// TIA Portal project "红黄绿等" (V16)

(* hardware
DEVICE "HMI_1"  KTP700 Basic PN
   slot 0: "HMI_1"  KTP700 Basic PN  6AV2 123-2GB03-0AX0  16.0.0.0
   slot 1: "HMI_RT_1"  KTP700 Basic PN  6AV2 123-2GB03-0AX0  16.0.0.0
   slot 5: "HMI_1.IE_CP_1"  PROFINET Interface  16.0.0.0
      slot 1: "PROFINET Interface_1"  PROFINET Interface
         slot 1: "Port_1"  Port
DEVICE "S7-1200 station_1"  S7-1200 Station
   slot 0: "Rack_0"  S7-1200 Rack  Rack  V1.0
   slot 1: "PLC_1"  CPU 1212C DC/DC/DC  6ES7 212-1AE40-0XB0  V4.2
   slot 2: "DI 16/DQ 16x24VDC_1"  6ES7 223-1BL32-0XB0  V2.0
DEVICE "S7-1200 station_2"  S7-1200 Station
   slot 0: "Rack_0"  S7-1200 Rack  Rack  V1.0
   slot 1: "PLC_2"  CPU 1212C DC/DC/DC  6ES7 212-1AE40-0XB0  V4.2
   slot 2: "DI 16/DQ 16x24VDC_1"  6ES7 223-1BL32-0XB0  V2.0
*)

// ===== PLC "PLC_1"  CPU 1212C DC/DC/DC =====

VAR_GLOBAL   // PLC tag table "默认变量表"
   "System_Byte" AT %MB1 : Byte;
   "FirstScan" AT %M1.0 : Bool;
   "DiagStatusUpdate" AT %M1.1 : Bool;
   "AlwaysTRUE" AT %M1.2 : Bool;
   "AlwaysFALSE" AT %M1.3 : Bool;
   "Tag_1" AT %M8.1 : Bool;
   "Tag_3" AT %MD90 : Real;
   "Tag_4" AT %MD80 : Real;
END_VAR

VAR_GLOBAL   // PLC tag table "io表"
   "x轴脉冲" AT %Q0.0 : Bool;
   "x轴方向" AT %Q0.1 : Bool;
   "z轴脉冲" AT %Q0.2 : Bool;
   "z轴方向" AT %Q0.3 : Bool;
   "x轴前限位" AT %I0.0 : Bool;
   "x轴原点" AT %I0.1 : Bool;
   "x轴后限位" AT %I0.2 : Bool;
   "z轴上限位" AT %I0.3 : Bool;
   "z轴原点" AT %I0.4 : Bool;
   "z轴下限位" AT %I0.5 : Bool;
   "输送线A右传感器" AT %I1.0 : Bool;
   "输送线A左传感器" AT %I1.1 : Bool;
   "启动" AT %I1.4 : Bool;
   "复位" AT %I1.5 : Bool;
   "急停" AT %I1.6 : Bool;
   "单机/联动" AT %I1.7 : Bool;
   "旋转气缸左转" AT %I2.0 : Bool;
   "旋转气缸右转" AT %I2.1 : Bool;
   "伸出前限位" AT %I2.2 : Bool;
   "伸出后限位" AT %I2.3 : Bool;
   "黄灯" AT %Q1.0 : Bool;
   "红灯" AT %Q1.2 : Bool;
   "气缸左旋" AT %Q1.4 : Bool;
   "气缸右旋" AT %Q1.5 : Bool;
   "气缸伸缩" AT %Q1.6 : Bool;
   "气缸夹紧" AT %Q1.7 : Bool;
   "输送带A正转" AT %Q2.0 : Bool;
   "输送带A反转" AT %Q2.1 : Bool;
   "手自动切换" AT %M2.6 : Bool;
   "自动启动按钮" AT %M2.7 : Bool;
   "x轴前进-触点" AT %M6.0 : Bool;
   "x轴后退-触点" AT %M6.1 : Bool;
   "z轴下移-触点" AT %M6.2 : Bool;
   "z轴上移-触点" AT %M6.3 : Bool;
   "x轴前进" AT %M7.0 : Bool;
   "x轴后退" AT %M7.1 : Bool;
   "x轴回原点" AT %M7.2 : Bool;
   "z轴上移" AT %M7.3 : Bool;
   "z轴下移" AT %M7.4 : Bool;
   "z轴回原点" AT %M7.5 : Bool;
   "x轴启动标志位" AT %M2.0 : Bool;
   "x轴完成标志位" AT %M2.1 : Bool;
   "z轴启动标志位" AT %M2.2 : Bool;
   "z轴完成标志位" AT %M2.3 : Bool;
   "x轴回原点(1)" AT %M2.4 : Bool;
   "z轴回原点(1)" AT %M2.5 : Bool;
   "启动整个程序" AT %M5.0 : Bool;
   "tag_2" AT %M5.2 : Bool;
   "自动模式" AT %M5.3 : Bool;
   "x轴取料移动标志" AT %M3.0 : Bool;
   "tag_5" AT %M20.0 : Bool;
   "z轴取料移动标志位" AT %M3.1 : Bool;
   "tag_7" AT %M20.1 : Bool;
   "x轴定位数据" AT %MD30 : Real;
   "z轴定位数据" AT %MD40 : Real;
   "启动气缸左旋标志位" AT %M3.2 : Bool;
   "启动气缸伸缩标志位" AT %M3.3 : Bool;
   "启动气缸夹取标志位" AT %M3.4 : Bool;
   "z轴上升标志位" AT %M3.5 : Bool;
   "tag_12" AT %M20.2 : Bool;
   "气缸回缩标志位" AT %M3.6 : Bool;
   "气缸右旋标志位" AT %M3.7 : Bool;
   "x轴启动放料位" AT %M4.0 : Bool;
   "tag_16" AT %M20.3 : Bool;
   "z轴上升到放料位" AT %M4.1 : Bool;
   "tag_18" AT %M20.4 : Bool;
   "气缸伸出放料标志位" AT %M4.2 : Bool;
   "气缸放松放料标志位" AT %M4.3 : Bool;
   "tag_21" AT %M4.4 : Bool;
   "X轴报错复位" AT %M7.6 : Bool;
   "z轴报错复位" AT %M7.7 : Bool;
   "tag_22" AT %MD50 : Real;
   "tag_23" AT %MD60 : Real;
   "tag_24" AT %MD70 : Real;
   "绿灯" AT %Q1.1 : Bool;
END_VAR

// folder: System blocks/Program resources

DATA_BLOCK "T1"   // DB3
{ S7_Optimized_Access := 'TRUE' }
AUTHOR : Simatic
FAMILY : IEC
NAME : IEC_TMR
VERSION : 1.0
// stored: InstanceOfName IEC_TIMER
"IEC_TIMER"
BEGIN
END_DATA_BLOCK

DATA_BLOCK "T2"   // DB4
{ S7_Optimized_Access := 'TRUE' }
AUTHOR : Simatic
FAMILY : IEC
NAME : IEC_TMR
VERSION : 1.0
// stored: InstanceOfName IEC_TIMER
"IEC_TIMER"
BEGIN
END_DATA_BLOCK

DATA_BLOCK "T3"   // DB5
{ S7_Optimized_Access := 'TRUE' }
AUTHOR : Simatic
FAMILY : IEC
NAME : IEC_TMR
VERSION : 1.0
// stored: InstanceOfName IEC_TIMER
"IEC_TIMER"
BEGIN
END_DATA_BLOCK

DATA_BLOCK "T4"   // DB6
{ S7_Optimized_Access := 'TRUE' }
AUTHOR : Simatic
FAMILY : IEC
NAME : IEC_TMR
VERSION : 1.0
// stored: InstanceOfName IEC_TIMER
"IEC_TIMER"
BEGIN
END_DATA_BLOCK

DATA_BLOCK "T5"   // DB7
{ S7_Optimized_Access := 'TRUE' }
AUTHOR : Simatic
FAMILY : IEC
NAME : IEC_TMR
VERSION : 1.0
// stored: InstanceOfName IEC_TIMER
"IEC_TIMER"
BEGIN
END_DATA_BLOCK

DATA_BLOCK "T7"   // DB8
{ S7_Optimized_Access := 'TRUE' }
AUTHOR : Simatic
FAMILY : IEC
NAME : IEC_TMR
VERSION : 1.0
// stored: InstanceOfName IEC_TIMER
"IEC_TIMER"
BEGIN
END_DATA_BLOCK

DATA_BLOCK "T6"   // DB9
{ S7_Optimized_Access := 'TRUE' }
AUTHOR : Simatic
FAMILY : IEC
NAME : IEC_TMR
VERSION : 1.0
// stored: InstanceOfName IEC_TIMER
"IEC_TIMER"
BEGIN
END_DATA_BLOCK

DATA_BLOCK "T8"   // DB10
{ S7_Optimized_Access := 'TRUE' }
AUTHOR : Simatic
FAMILY : IEC
NAME : IEC_TMR
VERSION : 1.0
// stored: InstanceOfName IEC_TIMER
"IEC_TIMER"
BEGIN
END_DATA_BLOCK

DATA_BLOCK "T9"   // DB11
{ S7_Optimized_Access := 'TRUE' }
AUTHOR : Simatic
FAMILY : IEC
NAME : IEC_TMR
VERSION : 1.0
// stored: InstanceOfName IEC_TIMER
"IEC_TIMER"
BEGIN
END_DATA_BLOCK

DATA_BLOCK "T10"   // DB12
{ S7_Optimized_Access := 'TRUE' }
AUTHOR : Simatic
FAMILY : IEC
NAME : IEC_TMR
VERSION : 1.0
// stored: InstanceOfName IEC_TIMER
"IEC_TIMER"
BEGIN
END_DATA_BLOCK

DATA_BLOCK "T11"   // DB13
{ S7_Optimized_Access := 'TRUE' }
AUTHOR : Simatic
FAMILY : IEC
NAME : IEC_TMR
VERSION : 1.0
// stored: InstanceOfName IEC_TIMER
"IEC_TIMER"
BEGIN
END_DATA_BLOCK

DATA_BLOCK "T12"   // DB14
{ S7_Optimized_Access := 'TRUE' }
AUTHOR : Simatic
FAMILY : IEC
NAME : IEC_TMR
VERSION : 1.0
// stored: InstanceOfName IEC_TIMER
"IEC_TIMER"
BEGIN
END_DATA_BLOCK

DATA_BLOCK "T13"   // DB15
{ S7_Optimized_Access := 'TRUE' }
AUTHOR : Simatic
FAMILY : IEC
NAME : IEC_TMR
VERSION : 1.0
// stored: InstanceOfName IEC_TIMER
"IEC_TIMER"
BEGIN
END_DATA_BLOCK

DATA_BLOCK "IEC_Timer_0_DB"   // DB28
{ S7_Optimized_Access := 'TRUE' }
AUTHOR : Simatic
FAMILY : IEC
NAME : IEC_TMR
VERSION : 1.0
// stored: InstanceOfName IEC_TIMER
"IEC_TIMER"
BEGIN
END_DATA_BLOCK

// folder: (top level)

DATA_BLOCK "轴_1"   // DB1, Motion_DB
{ S7_Optimized_Access := 'TRUE' }
AUTHOR : SIMATIC
FAMILY : BasicMC
NAME : TO_PosAx
VERSION : 6.0
// stored: InstanceOfName TO_PositioningAxis
"TO_PositioningAxis"
BEGIN
   // Axis.HomingReferencePointSwitch_AddressCU = %I0.1
   // Axis.LengthUnitNormalized.Distance = 1013
   // Axis.PositionLimitsMax_AddressCU = %I0.2
   // Axis.PositionLimitsMin_AddressCU = %I0.0
   // Axis.DirectionOutputEnabledCU = TRUE
   // Axis.OnlinePtoModeCU = 16#0000_0002
   // Axis.SelectedChannel2EnumCU = %Q0.1
   // Axis.SelectedChannel1EnumCU = %Q0.0
   // Pulse.MinDeltaDeltaFrequencyCU = 0.004
   // Pulse.MaxDeltaDeltaFrequencyCU = 1.0E+10
   // Pulse.MinDeltaFrequencyCU = 0.005
   // Pulse.MaxDeltaFrequencyCU = 9.5E+9
   // Pulse.MinFrequencyCU = 1.0
   // Pulse.MaxFrequencyCU = 100000.0
   // Pulse.OutputSourceCU = 16#0000_0000
   // Axis.SelectPTO = 0
END_DATA_BLOCK

DATA_BLOCK "轴_2"   // DB2, Motion_DB
{ S7_Optimized_Access := 'TRUE' }
AUTHOR : SIMATIC
FAMILY : BasicMC
NAME : TO_PosAx
VERSION : 6.0
// stored: InstanceOfName TO_PositioningAxis
"TO_PositioningAxis"
BEGIN
   // Axis.HomingReferencePointSwitch_AddressCU = %I0.4
   // Axis.LengthUnitNormalized.Distance = 1013
   // Axis.PositionLimitsMax_AddressCU = %I0.5
   // Axis.PositionLimitsMin_AddressCU = %I0.3
   // Axis.DirectionOutputEnabledCU = TRUE
   // Axis.OnlinePtoModeCU = 16#0000_0002
   // Axis.SelectedChannel2EnumCU = %Q0.3
   // Axis.SelectedChannel1EnumCU = %Q0.2
   // Pulse.MinDeltaDeltaFrequencyCU = 0.004
   // Pulse.MaxDeltaDeltaFrequencyCU = 1.0E+10
   // Pulse.MinDeltaFrequencyCU = 0.005
   // Pulse.MaxDeltaFrequencyCU = 9.5E+9
   // Pulse.MinFrequencyCU = 1.0
   // Pulse.MaxFrequencyCU = 100000.0
   // Pulse.OutputSourceCU = 16#0000_0000
   // Axis.SelectPTO = 1
   // Axis.OnlinePtoIndexCU = 1
END_DATA_BLOCK

FUNCTION "电机运转" : Void   // FC1, LAD
{ S7_Optimized_Access := 'TRUE' }
VERSION : 0.1
BEGIN

REGION Network 1: 启动两个电机轴
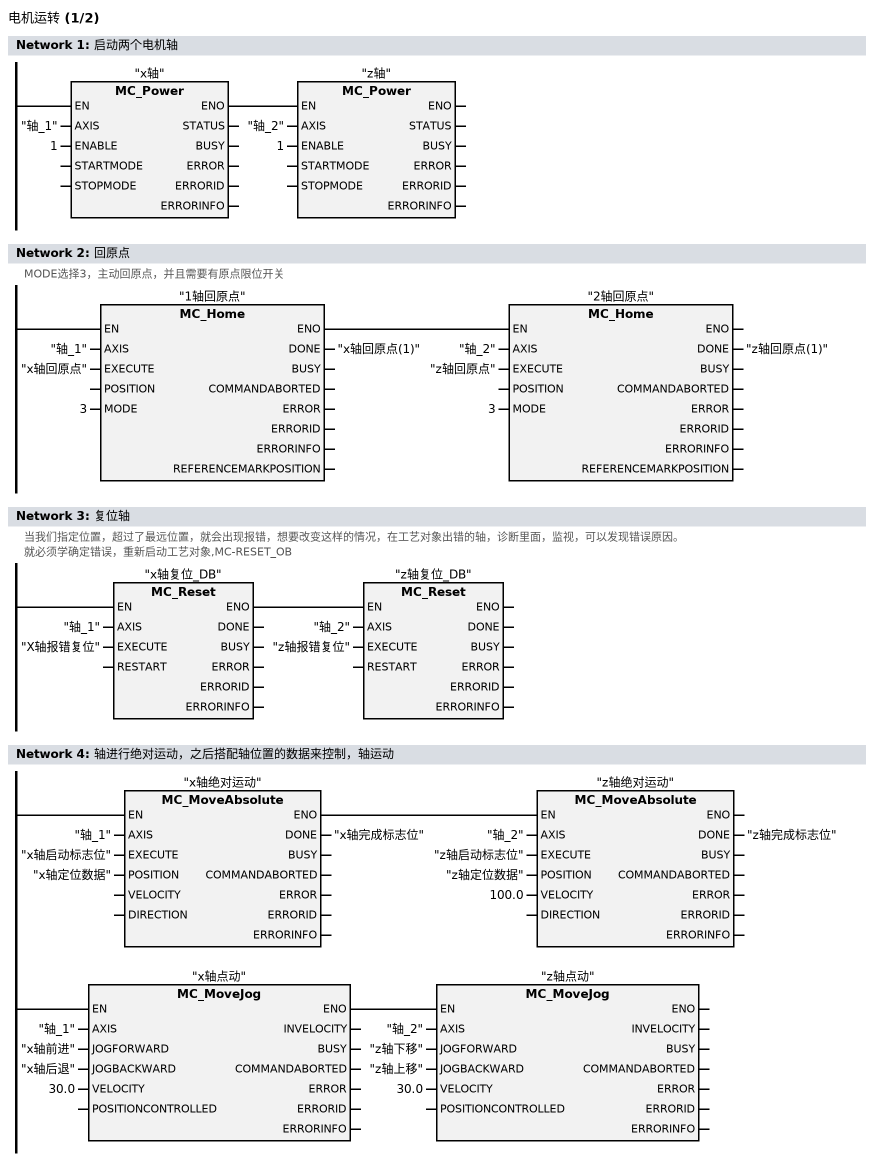
   // ENO of a box is taken as its EN; it also drops when the box reports an error
   "x轴"(Axis := "轴_1", Enable := 1);   // MC_Power
   "z轴"(Axis := "轴_2", Enable := 1);   // MC_Power
END_REGION

REGION Network 2: 回原点
   // MODE选择3，主动回原点，并且需要有原点限位开关
   // ENO of a box is taken as its EN; it also drops when the box reports an error
   "1轴回原点"(Axis := "轴_1", Execute := "x轴回原点", Mode := 3, Done => "x轴回原点(1)");   // MC_Home
   "2轴回原点"(Axis := "轴_2", Execute := "z轴回原点", Mode := 3, Done => "z轴回原点(1)");   // MC_Home
END_REGION

REGION Network 3: 复位轴
   // 当我们指定位置，超过了最远位置，就会出现报错，想要改变这样的情况，在工艺对象出错的轴，诊断里面，监视，可以发现错误原因。
   // 就必须学确定错误，重新启动工艺对象,MC-RESET_OB
   // ENO of a box is taken as its EN; it also drops when the box reports an error
   "x轴复位_DB"(Axis := "轴_1", Execute := "X轴报错复位");   // MC_Reset
   "z轴复位_DB"(Axis := "轴_2", Execute := "z轴报错复位");   // MC_Reset
END_REGION

REGION Network 4: 轴进行绝对运动，之后搭配轴位置的数据来控制，轴运动
   // ENO of a box is taken as its EN; it also drops when the box reports an error
   "x轴绝对运动"(Axis := "轴_1", Execute := "x轴启动标志位", Position := "x轴定位数据", Done => "x轴完成标志位");   // MC_MoveAbsolute
   "z轴绝对运动"(Axis := "轴_2", Execute := "z轴启动标志位", Position := "z轴定位数据", Velocity := 100.0, Done => "z轴完成标志位");   // MC_MoveAbsolute
   "x轴点动"(Axis := "轴_1", JogForward := "x轴前进", JogBackward := "x轴后退", Velocity := 30.0);   // MC_MoveJog
   "z轴点动"(Axis := "轴_2", JogForward := "z轴下移", JogBackward := "z轴上移", Velocity := 30.0);   // MC_MoveJog
END_REGION

REGION Network 5
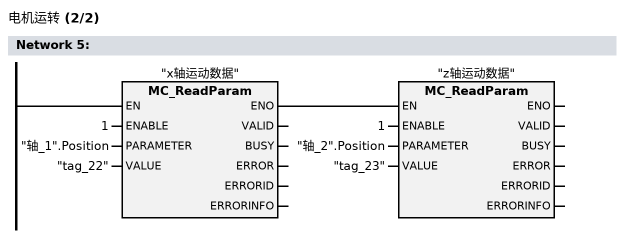
   // ENO of a box is taken as its EN; it also drops when the box reports an error
   "x轴运动数据"(Enable := 1, Parameter := "轴_1".Position, Value := "tag_22");   // MC_ReadParam
   "z轴运动数据"(Enable := 1, Parameter := "轴_2".Position, Value := "tag_23");   // MC_ReadParam
END_REGION
END_FUNCTION

ORGANIZATION_BLOCK "Main"   // OB1, LAD, ProgramCycle
TITLE = "Main Program Sweep (Cycle)"
{ S7_Optimized_Access := 'TRUE' }
VERSION : 0.1
   VAR_INPUT
      Initial_Call : Bool;   // Initial call of this OB
      Remanence : Bool;   // =True, if remanent data are available
   END_VAR
   VAR_TEMP   // added for the SCL form of the ladder/FBD networks
      _w1 : Bool;
      _w2 : Bool;
      _w3 : Bool;
   END_VAR
BEGIN

REGION Network 1: 初始化程序，并且启动程序
   // 利用M1.0达到首次循环，启动复位
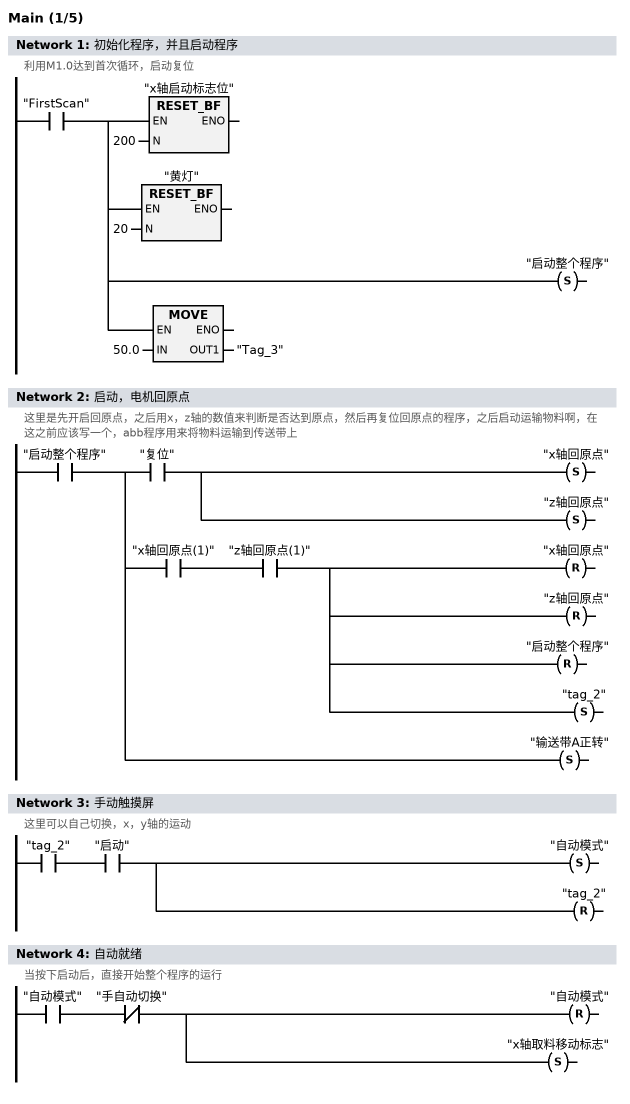
   // no SCL statement known for RBitfield: written as a call
   #_w1 := "FirstScan";
   IF #_w1 THEN
       RESET_BF(operand := "x轴启动标志位", n := 200);
       RESET_BF(operand := "黄灯", n := 20);
       "启动整个程序" := TRUE;
       "Tag_3" := 50.0;
   END_IF;
END_REGION

REGION Network 2: 启动，电机回原点
   // 这里是先开启回原点，之后用x，z轴的数值来判断是否达到原点，然后再复位回原点的程序，之后启动运输物料啊，在这之前应该写一个，abb程序用来将物料运输到传送带上
   RUNG wire#powerrail
      Contact( "启动整个程序" )
      wire#w1
      Contact( "复位" )
      wire#w2
      S_Coil( "x轴回原点" )
   END_RUNG
   RUNG wire#w2
      S_Coil( "z轴回原点" )
   END_RUNG
   RUNG wire#w1
      Contact( "x轴回原点(1)" )
      Contact( "z轴回原点(1)" )
      wire#w3
      R_Coil( "x轴回原点" )
   END_RUNG
   RUNG wire#w3
      R_Coil( "z轴回原点" )
   END_RUNG
   RUNG wire#w3
      R_Coil( "启动整个程序" )
   END_RUNG
   RUNG wire#w3
      S_Coil( "tag_2" )
   END_RUNG
   RUNG wire#w1
      S_Coil( "输送带A正转" )
   END_RUNG
   // the same network as SCL:
   IF "启动整个程序" AND "复位" THEN
       "x轴回原点" := TRUE;
       "z轴回原点" := TRUE;
   END_IF;
   IF "启动整个程序" AND "x轴回原点(1)" AND "z轴回原点(1)" THEN
       "x轴回原点" := FALSE;
       "z轴回原点" := FALSE;
   END_IF;
   #_w1 := "启动整个程序";
   #_w2 := "启动整个程序" AND "x轴回原点(1)" AND "z轴回原点(1)";
   IF #_w2 THEN
       "启动整个程序" := FALSE;
       "tag_2" := TRUE;
   END_IF;
   IF #_w1 THEN "输送带A正转" := TRUE; END_IF;
END_REGION

REGION Network 3: 手动触摸屏
   // 这里可以自己切换，x，y轴的运动
   RUNG wire#powerrail
      Contact( "tag_2" )
      Contact( "启动" )
      wire#w1
      S_Coil( "自动模式" )
   END_RUNG
   RUNG wire#w1
      R_Coil( "tag_2" )
   END_RUNG
   // the same network as SCL:
   IF "tag_2" AND "启动" THEN
       "自动模式" := TRUE;
       "tag_2" := FALSE;
   END_IF;
END_REGION

REGION Network 4: 自动就绪
   // 当按下启动后，直接开始整个程序的运行
   RUNG wire#powerrail
      Contact( "自动模式" )
      I_Contact( "手自动切换" )
      wire#w1
      R_Coil( "自动模式" )
   END_RUNG
   RUNG wire#w1
      S_Coil( "x轴取料移动标志" )
   END_RUNG
   // the same network as SCL:
   #_w1 := "自动模式" AND NOT "手自动切换";
   IF #_w1 THEN
       "自动模式" := FALSE;
       "x轴取料移动标志" := TRUE;
   END_IF;
END_REGION

REGION Network 5: x轴取料
   // 此处对应传送带上的传感器，限位开关感应到物料,，输送带停止输送
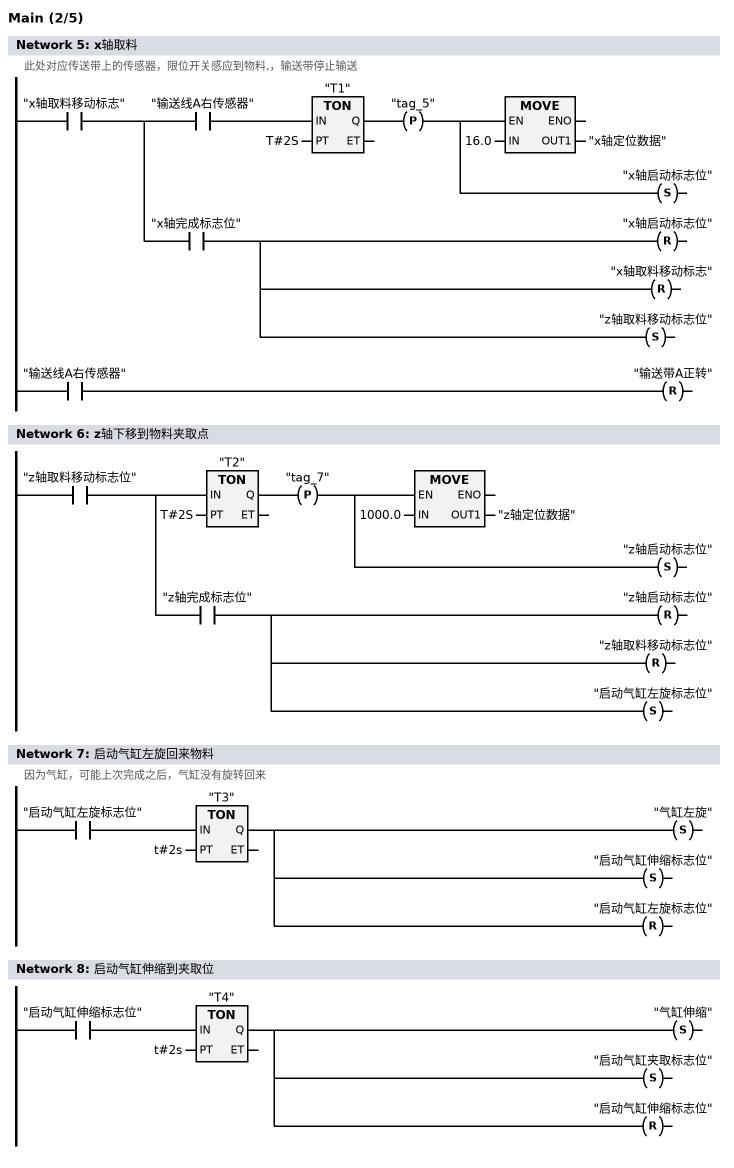
   "T1".TON(IN := "x轴取料移动标志" AND "输送线A右传感器", PT := T#2S);
   #_w1 := "T1".Q AND NOT "tag_5";   // rising edge
   "tag_5" := "T1".Q;
   IF #_w1 THEN
       "x轴定位数据" := 16.0;
       "x轴启动标志位" := TRUE;
   END_IF;
   IF "x轴取料移动标志" AND "x轴完成标志位" THEN "x轴启动标志位" := FALSE; END_IF;
   #_w2 := "x轴取料移动标志" AND "x轴完成标志位";
   IF #_w2 THEN
       "x轴取料移动标志" := FALSE;
       "z轴取料移动标志位" := TRUE;
   END_IF;
   IF "输送线A右传感器" THEN "输送带A正转" := FALSE; END_IF;
END_REGION

REGION Network 6: z轴下移到物料夹取点
   "T2".TON(IN := "z轴取料移动标志位", PT := T#2S);
   #_w1 := "T2".Q AND NOT "tag_7";   // rising edge
   "tag_7" := "T2".Q;
   IF #_w1 THEN
       "z轴定位数据" := 1000.0;
       "z轴启动标志位" := TRUE;
   END_IF;
   IF "z轴取料移动标志位" AND "z轴完成标志位" THEN "z轴启动标志位" := FALSE; END_IF;
   #_w2 := "z轴取料移动标志位" AND "z轴完成标志位";
   IF #_w2 THEN
       "z轴取料移动标志位" := FALSE;
       "启动气缸左旋标志位" := TRUE;
   END_IF;
END_REGION

REGION Network 7: 启动气缸左旋回来物料
   // 因为气缸，可能上次完成之后，气缸没有旋转回来
   "T3".TON(IN := "启动气缸左旋标志位", PT := t#2s);
   IF "T3".Q THEN
       "气缸左旋" := TRUE;
       "启动气缸伸缩标志位" := TRUE;
       "启动气缸左旋标志位" := FALSE;
   END_IF;
END_REGION

REGION Network 8: 启动气缸伸缩到夹取位
   "T4".TON(IN := "启动气缸伸缩标志位", PT := t#2s);
   IF "T4".Q THEN
       "气缸伸缩" := TRUE;
       "启动气缸夹取标志位" := TRUE;
       "启动气缸伸缩标志位" := FALSE;
   END_IF;
END_REGION

REGION Network 9: 启动气缸夹取
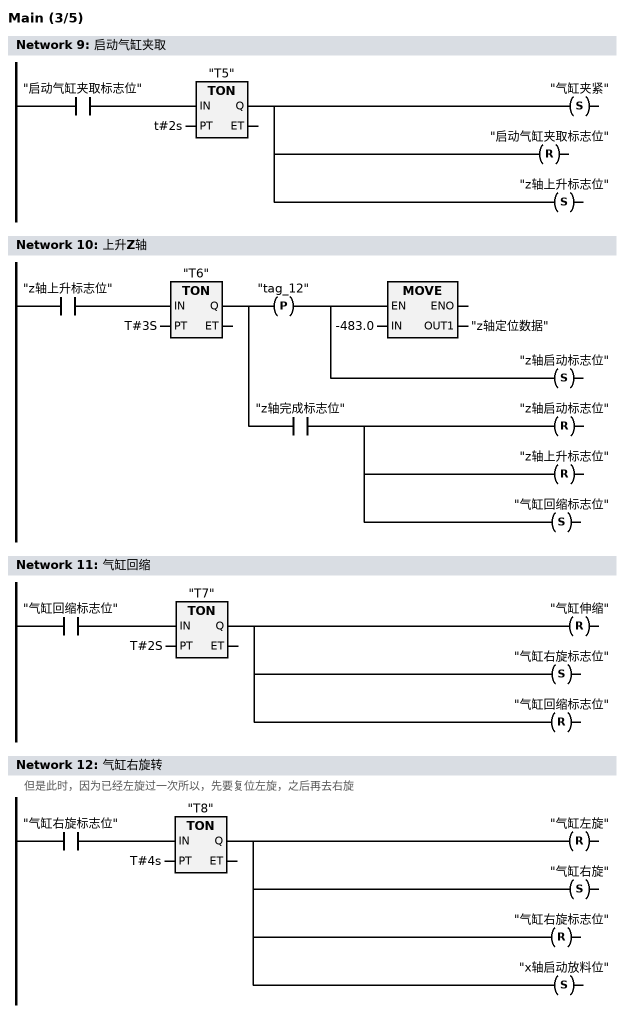
   "T5".TON(IN := "启动气缸夹取标志位", PT := t#2s);
   IF "T5".Q THEN
       "气缸夹紧" := TRUE;
       "启动气缸夹取标志位" := FALSE;
       "z轴上升标志位" := TRUE;
   END_IF;
END_REGION

REGION Network 10: 上升Z轴
   "T6".TON(IN := "z轴上升标志位", PT := T#3S);
   #_w1 := "T6".Q AND NOT "tag_12";   // rising edge
   "tag_12" := "T6".Q;
   IF #_w1 THEN
       "z轴定位数据" := -483.0;
       "z轴启动标志位" := TRUE;
   END_IF;
   IF "T6".Q AND "z轴完成标志位" THEN
       "z轴启动标志位" := FALSE;
       "z轴上升标志位" := FALSE;
       "气缸回缩标志位" := TRUE;
   END_IF;
END_REGION

REGION Network 11: 气缸回缩
   "T7".TON(IN := "气缸回缩标志位", PT := T#2S);
   IF "T7".Q THEN
       "气缸伸缩" := FALSE;
       "气缸右旋标志位" := TRUE;
       "气缸回缩标志位" := FALSE;
   END_IF;
END_REGION

REGION Network 12: 气缸右旋转
   // 但是此时，因为已经左旋过一次所以，先要复位左旋，之后再去右旋
   "T8".TON(IN := "气缸右旋标志位", PT := T#4s);
   IF "T8".Q THEN
       "气缸左旋" := FALSE;
       "气缸右旋" := TRUE;
       "气缸右旋标志位" := FALSE;
       "x轴启动放料位" := TRUE;
   END_IF;
END_REGION

REGION Network 13: x轴移动到放料位
   // 我对于x轴来说，每排放3个，
   // 所以当我想要进行循环的时候，我可以写一个递增的数据，每当x移动3次之后
   // 就在z轴上升的程序里面，进行一次加法/减法计算
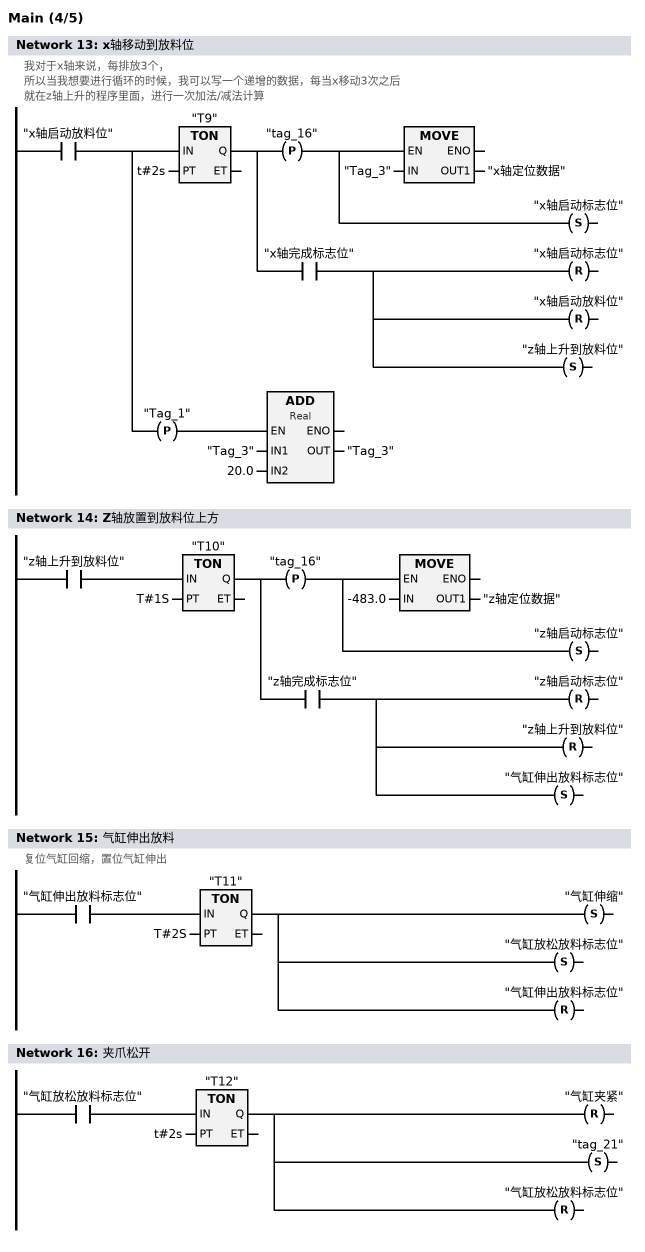
   "T9".TON(IN := "x轴启动放料位", PT := t#2s);
   #_w1 := "T9".Q AND NOT "tag_16";   // rising edge
   "tag_16" := "T9".Q;
   IF #_w1 THEN
       "x轴定位数据" := "Tag_3";
       "x轴启动标志位" := TRUE;
   END_IF;
   IF "T9".Q AND "x轴完成标志位" THEN "x轴启动标志位" := FALSE; END_IF;
   #_w2 := "x轴启动放料位";
   IF "T9".Q AND "x轴完成标志位" THEN
       "x轴启动放料位" := FALSE;
       "z轴上升到放料位" := TRUE;
   END_IF;
   #_w3 := #_w2 AND NOT "Tag_1";   // rising edge
   "Tag_1" := #_w2;
   IF #_w3 THEN "Tag_3" := "Tag_3" + 20.0; END_IF;
END_REGION

REGION Network 14: Z轴放置到放料位上方
   "T10".TON(IN := "z轴上升到放料位", PT := T#1S);
   #_w1 := "T10".Q AND NOT "tag_16";   // rising edge
   "tag_16" := "T10".Q;
   IF #_w1 THEN
       "z轴定位数据" := -483.0;
       "z轴启动标志位" := TRUE;
   END_IF;
   IF "T10".Q AND "z轴完成标志位" THEN
       "z轴启动标志位" := FALSE;
       "z轴上升到放料位" := FALSE;
       "气缸伸出放料标志位" := TRUE;
   END_IF;
END_REGION

REGION Network 15: 气缸伸出放料
   // 复位气缸回缩，置位气缸伸出
   "T11".TON(IN := "气缸伸出放料标志位", PT := T#2S);
   IF "T11".Q THEN
       "气缸伸缩" := TRUE;
       "气缸放松放料标志位" := TRUE;
       "气缸伸出放料标志位" := FALSE;
   END_IF;
END_REGION

REGION Network 16: 夹爪松开
   "T12".TON(IN := "气缸放松放料标志位", PT := t#2s);
   IF "T12".Q THEN
       "气缸夹紧" := FALSE;
       "tag_21" := TRUE;
       "气缸放松放料标志位" := FALSE;
   END_IF;
END_REGION

REGION Network 17: 结束复位
   // 如果要进行循环，此处应该重新置位
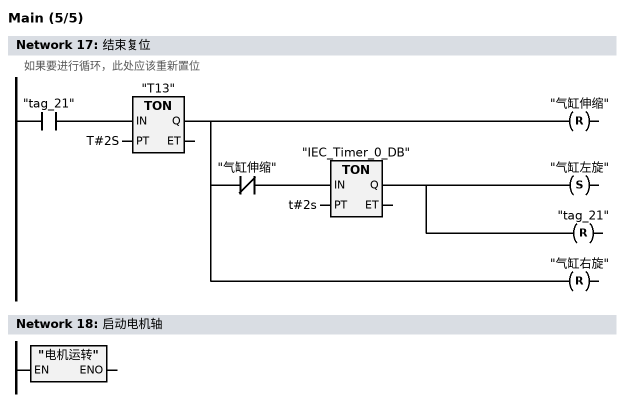
   "T13".TON(IN := "tag_21", PT := T#2S);
   IF "T13".Q THEN "气缸伸缩" := FALSE; END_IF;
   "IEC_Timer_0_DB".TON(IN := "T13".Q AND NOT "气缸伸缩", PT := t#2s);
   IF "IEC_Timer_0_DB".Q THEN
       "气缸左旋" := TRUE;
       "tag_21" := FALSE;
   END_IF;
   IF "T13".Q THEN "气缸右旋" := FALSE; END_IF;
END_REGION

REGION Network 18: 启动电机轴
   RUNG wire#powerrail
      "电机运转"()
   END_RUNG
   // the same network as SCL:
   "电机运转"();
END_REGION
END_ORGANIZATION_BLOCK

// ===== PLC "PLC_2"  CPU 1212C DC/DC/DC =====

VAR_GLOBAL   // PLC tag table "默认变量表"
   "Tag_1" AT %I1.4 : Bool;
   "Tag_2" AT %I1.5 : Bool;
   "Tag_3" AT %Q1.1 : Bool;
   "x轴脉冲" AT %Q0.0 : Bool;
   "x轴方向" AT %Q0.1 : Bool;
   "轴_1_LowHwLimitSwitch" AT %I0.0 : Bool;
   "轴_1_HighHwLimitSwitch" AT %I0.2 : Bool;
   "轴_1_归位开关" AT %I0.1 : Bool;
   "z轴脉冲" AT %Q0.2 : Bool;
   "z轴方向" AT %Q0.3 : Bool;
   "轴_2_LowHwLimitSwitch" AT %I0.3 : Bool;
   "轴_2_HighHwLimitSwitch" AT %I0.5 : Bool;
   "轴_2_归位开关" AT %I0.4 : Bool;
END_VAR

ORGANIZATION_BLOCK "Main"   // OB1, LAD, ProgramCycle
TITLE = "Main Program Sweep (Cycle)"
{ S7_Optimized_Access := 'TRUE' }
VERSION : 0.1
   VAR_INPUT
      Initial_Call : Bool;   // Initial call of this OB
      Remanence : Bool;   // =True, if remanent data are available
   END_VAR
BEGIN

REGION Network 1
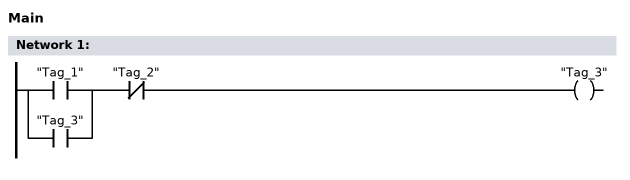
   RUNG wire#powerrail
      Contact( "Tag_1" )
      wire#w1
      I_Contact( "Tag_2" )
      Coil( "Tag_3" )
   END_RUNG
   RUNG wire#powerrail
      Contact( "Tag_3" )
   END_RUNG wire#w1
   // the same network as SCL:
   "Tag_3" := ("Tag_1" OR "Tag_3") AND NOT "Tag_2";
END_REGION
END_ORGANIZATION_BLOCK

(* ===== HMI "HMI_RT_1" =====
system functions are stored by id; their names below are inferred from use
connection "HMI_连接_1": ETHERNET, SMART_S7_1200_OMS

HMI tags "默认变量表"
   "Tag_ScreenNumber" : UInt, internal
   "启动" : Bool = PLC 启动 AT %I1.4, 1 s
   "停止" : Bool = PLC 停止 AT %M2.1, 1 s
   "东西绿" : Bool = PLC 东西绿 AT %Q0.0, 1 s
   "东西黄" : Bool = PLC 东西黄 AT %Q0.1, 1 s
   "东西红" : Bool = PLC 东西红 AT %Q0.2, 1 s
   "南北绿" : Bool = PLC 南北绿 AT %Q0.3, 1 s
   "南北红" : Bool = PLC 南北红 AT %Q0.5, 1 s
   "南北黄" : Bool = PLC 南北黄 AT %Q0.4, 1 s

Template "模板_1" 800x480
   Button "退出" at 714,429 size 71x50; TextOff '退出'; PictureOff "ExitRuntime_KTP700_Basic_PN_TR"; PictureOn "ExitRuntime_KTP700_Basic_PN_TR"
      on Release: StopRuntime(0)
   Button "Template_Button" at 614,429 size 71x50; TextOff 'Text'
   Button "Template_Button_1" at 514,429 size 71x50; TextOff 'Text'
   Button "Template_Button_2" at 414,429 size 71x50; TextOff 'Text'
   Button "Template_Button_3" at 314,429 size 71x50; TextOff 'Text'
   Button "Template_Button_4" at 214,429 size 71x50; TextOff 'Text'
   Button "Template_Button_5" at 114,429 size 71x50; TextOff 'Text'
   Button "起始画面" at 14,429 size 71x50; TextOff '起始画面'; PictureOff "NavigateHome_KTP700_Basic_PN_TR"; PictureOn "NavigateHome_KTP700_Basic_PN_TR"
      on Release: ActivateScreen("根画面", 0)
   SymbolicIOField "Symbolic_IO_Field_Screen" at 93,9 size 600x33; TextOff '0'; TextOn '1'; TextList "TextList_ScreenNames"
      ProcessValue <- "Tag_ScreenNumber"
      on Change: ActivateScreenByNumber("Tag_ScreenNumber", 0)
   DateTimeField "HmiScreenItemData" at 695,25 size 105x25
   DateTimeField "HmiScreenItemData_1" at 695,0 size 105x25
   GraphicView "Logo" at 0,0 size 91x51; Picture "HMI_1 的 Logo"

screen "根画面" 800x480, template "模板_1"
   on GenerateScreen: SetTag("Tag_ScreenNumber", 1)
   Button "按钮_1" at 199,244 size 96x32; TextOff '启动'
      on Press: SetBit("启动")
      on Release: ResetBit("启动")
   Circle "圆_1" at 392,99 size 48x48
      Appearance <- "东西红"
   TextField "文本域_1" at 385,62 size 71x37; Text '东西'
   TextField "文本域_2" at 542,59 size 71x37; Text '南北'
   Circle "圆_2" at 548,101 size 48x48
      Appearance <- "南北绿"
   Button "按钮_2" at 408,245 size 96x32; TextOff '停止'
      on Release: ResetBit("停止")
      on Press: SetBit("停止")
   Circle "圆_3" at 306,99 size 48x48
      Appearance <- "东西黄"
   Circle "圆_4" at 219,101 size 48x48
      Appearance <- "东西绿"
   Circle "圆_5" at 622,99 size 48x48
      Appearance <- "南北红"
   Circle "圆_6" at 708,101 size 48x48
      Appearance <- "南北黄"
*)